KUKA KRL program: ab_st600_r1.src, ab_st600_r1.dat

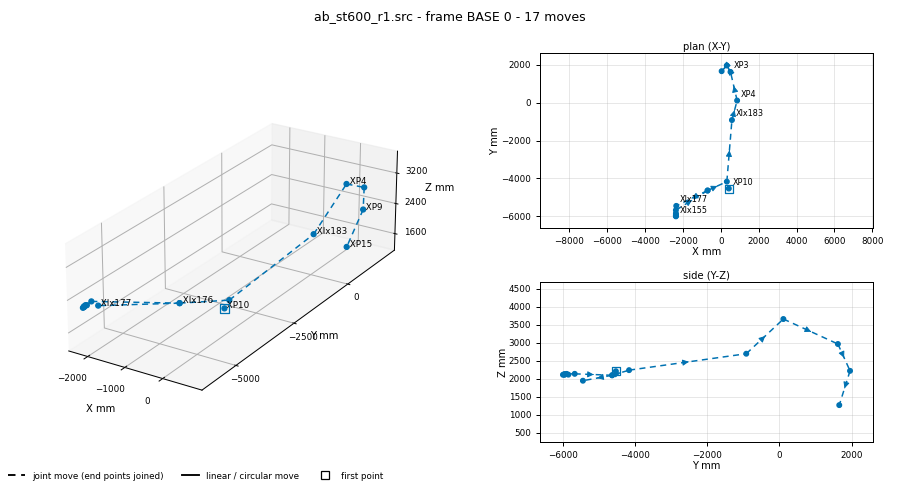
[picture p0: tool path of ab_st600_r1.src in frame BASE 0, 17 of 22 moves have a stored position in this frame; points joined in program order, loops and branches not executed]
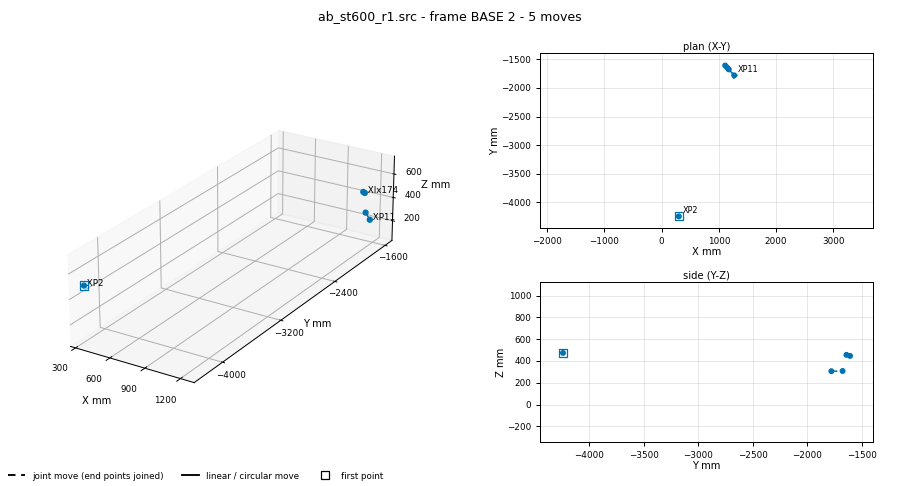
[picture p1: tool path of ab_st600_r1.src in frame BASE 2, 5 of 22 moves have a stored position in this frame; points joined in program order, loops and branches not executed]
--- ab_st600_r1.src ---
&ACCESS RVP1
&REL 63
&COMMENT Deposita traseira ACCELO
&PARAM DISKPATH = KRC:\R1\Program\MANIPULACAO LTC
&PARAM TEMPLATE = C:\KRC\Roboter\Template\vorgabe
&PARAM EDITMASK = *
DEF ab_st600_r1( )
;FOLD INI
  ;FOLD BASISTECH INI
    GLOBAL INTERRUPT DECL 3 WHEN $STOPMESS==TRUE DO IR_STOPM ( )
    INTERRUPT ON 3
    BAS (#INITMOV,0 )
  ;ENDFOLD (BASISTECH INI)
;FOLD GRIPPERTECH INI
USER_GRP(0,DUMMY,DUMMY,GDEFAULT)
;ENDFOLD (GRIPPERTECH INI)
  ;FOLD USER INI
    ;Make your modifications here

  ;ENDFOLD (USER INI)
;ENDFOLD (INI)

; Caracterização dos meios de produção:
; Versão Atual:
; 08/06/2013 12:00 Name: P13.050-R1 CHANGES: Deposita Traseira
; Accelo na Geobox

chk_w7_wechs_ok ( )              ; CHECK GRIPPER TRASEIRO


;FOLD PTP P10 Vel=100 % PDAT30 Tool[7]:Painel Traseiro Accelo Base[0];%{PE}%R 8.2.20,%MKUKATPBASIS,%CMOVE,%VPTP,%P 1:PTP, 2:P10, 3:, 5:100, 7:PDAT30
$BWDSTART=FALSE
PDAT_ACT=PPDAT30
FDAT_ACT=FP10
BAS(#PTP_PARAMS,100)
PTP XP10
;ENDFOLD

;FOLD PTP P2 Vel=100 % PDAT20 Tool[7]:Painel Traseiro Accelo Base[2]:Accelo;%{PE}%R 8.2.20,%MKUKATPBASIS,%CMOVE,%VPTP,%P 1:PTP, 2:P2, 3:, 5:100, 7:PDAT20
$BWDSTART=FALSE
PDAT_ACT=PPDAT20
FDAT_ACT=FP2
BAS(#PTP_PARAMS,100)
PTP XP2
;ENDFOLD

;FOLD OUT 3346 'Entrega peça Geo box' State=TRUE ;%{PE}%R 8.2.20,%MKUKATPBASIS,%COUT,%VOUTX,%P 2:3346, 3:Entrega peça Geo box, 5:TRUE, 6:
$OUT[3346]=TRUE
;ENDFOLD
;FOLD WAIT FOR ( IN 3346 'Aguarda lib. Entregar peça Geo box' );%{PE}%R 8.2.20,%MKUKATPBASIS,%CEXT_WAIT_FOR,%VEXT_WAIT_FOR,%P 2:, 4:, 5:$IN, 6:3346, 7:Aguarda lib. Entregar peça Geo box, 9:
WAIT FOR  ( $IN[3346] )
;ENDFOLD
;FOLD OUT 3346 'Entrega peça Geo box' State=FALSE ;%{PE}%R 8.2.20,%MKUKATPBASIS,%COUT,%VOUTX,%P 2:3346, 3:Entrega peça Geo box, 5:FALSE, 6:
$OUT[3346]=FALSE
;ENDFOLD
;FOLD OUT 3344 'R1 entregou peça geo box' State=FALSE ;%{PE}%R 8.2.20,%MKUKATPBASIS,%COUT,%VOUTX,%P 2:3344, 3:R1 entregou peça geo box, 5:FALSE, 6:
$OUT[3344]=FALSE
;ENDFOLD

;FOLD Collision.Monitoring_AREA_5_On ;%{PE}%MKUKATPUSER
COLLSTOP( 11, 1 ) ;not Interrupt-Controlled
;ENDFOLD
;FOLD Collision.Monitoring_AREA_6_On ;%{PE}%MKUKATPUSER
COLLSTOP( 12, 1 ) ;not Interrupt-Controlled
;ENDFOLD

;FOLD OUT 3340 'AREA_CLEAR_AGV' State=FALSE ;%{PE}%R 8.2.20,%MKUKATPBASIS,%COUT,%VOUTX,%P 2:3340, 3:AREA_CLEAR_AGV, 5:FALSE, 6:
$OUT[3340]=FALSE
;ENDFOLD
;FOLD OUT 3348 'Fora area GEOBOX' State=FALSE ;%{PE}%R 8.2.20,%MKUKATPBASIS,%COUT,%VOUTX,%P 2:3348, 3:Fora area GEOBOX, 5:FALSE, 6:
$OUT[3348]=FALSE
;ENDFOLD

;FOLD PTP lx176 CONT Vel=100 % PDAT8 Tool[7]:Painel Traseiro Accelo Base[0];%{PE}%R 8.2.20,%MKUKATPBASIS,%CMOVE,%VPTP,%P 1:PTP, 2:lx176, 3:C_DIS, 5:100, 7:PDAT8
$BWDSTART=FALSE
PDAT_ACT=PPDAT8
FDAT_ACT=Flx176
BAS(#PTP_PARAMS,100)
PTP Xlx176 C_DIS
;ENDFOLD
;FOLD PTP lx177 CONT Vel=100 % PDAT9 Tool[7]:Painel Traseiro Accelo Base[0];%{PE}%R 8.2.20,%MKUKATPBASIS,%CMOVE,%VPTP,%P 1:PTP, 2:lx177, 3:C_DIS, 5:100, 7:PDAT9
$BWDSTART=FALSE
PDAT_ACT=PPDAT9
FDAT_ACT=Flx177
BAS(#PTP_PARAMS,100)
PTP Xlx177 C_DIS
;ENDFOLD

;FOLD PTP P11 Vel=100 % PDAT31 Tool[7]:Painel Traseiro Accelo Base[2]:Accelo;%{PE}%R 8.2.20,%MKUKATPBASIS,%CMOVE,%VPTP,%P 1:PTP, 2:P11, 3:, 5:100, 7:PDAT31
$BWDSTART=FALSE
PDAT_ACT=PPDAT31
FDAT_ACT=FP11
BAS(#PTP_PARAMS,100)
PTP XP11
;ENDFOLD




;FOLD PTP lx178 Vel=100 % PDAT10 Tool[7]:Painel Traseiro Accelo Base[2]:Accelo;%{PE}%R 8.2.20,%MKUKATPBASIS,%CMOVE,%VPTP,%P 1:PTP, 2:lx178, 3:, 5:100, 7:PDAT10
$BWDSTART=FALSE
PDAT_ACT=PPDAT10
FDAT_ACT=Flx178
BAS(#PTP_PARAMS,100)
PTP Xlx178
;ENDFOLD


;FOLD PTP lx179 CONT Vel=70 % PDAT11 Tool[7]:Painel Traseiro Accelo Base[0];%{PE}%R 8.2.20,%MKUKATPBASIS,%CMOVE,%VPTP,%P 1:PTP, 2:lx179, 3:C_DIS, 5:70, 7:PDAT11
$BWDSTART=FALSE
PDAT_ACT=PPDAT11
FDAT_ACT=Flx179
BAS(#PTP_PARAMS,70)
PTP Xlx179 C_DIS
;ENDFOLD

IF (NOT(GHOST())) THEN

;FOLD ; bloqueado na Folder;%{PE}%R 8.2.20,%MKUKATPBASIS,%CCOMMENT,%VNORMAL,%P 2:bloqueado  na  Folder
;ENDFOLD

ENDIF

;FOLD LIN lx174 CONT Vel=0.25 m/s CPDAT0 Tool[7]:Painel Traseiro Accelo Base[0];%{PE}%R 8.2.20,%MKUKATPBASIS,%CMOVE,%VLIN,%P 1:LIN, 2:lx174, 3:C_DIS C_DIS, 5:0.25, 7:CPDAT0
$BWDSTART=FALSE
LDAT_ACT=LCPDAT0
FDAT_ACT=Flx174
BAS(#CP_PARAMS,0.25)
LIN Xlx174 C_DIS C_DIS
;ENDFOLD
;FOLD LIN lx173 CONT Vel=0.25 m/s CPDAT1 Tool[7]:Painel Traseiro Accelo Base[0];%{PE}%R 8.2.20,%MKUKATPBASIS,%CMOVE,%VLIN,%P 1:LIN, 2:lx173, 3:C_DIS C_DIS, 5:0.25, 7:CPDAT1
$BWDSTART=FALSE
LDAT_ACT=LCPDAT1
FDAT_ACT=Flx173
BAS(#CP_PARAMS,0.25)
LIN Xlx173 C_DIS C_DIS
;ENDFOLD
;FOLD LIN P12 Vel=0.25 m/s CPDAT2 Tool[7]:Painel Traseiro Accelo Base[0];%{PE}%R 8.2.20,%MKUKATPBASIS,%CMOVE,%VLIN,%P 1:LIN, 2:P12, 3:, 5:0.25, 7:CPDAT2
$BWDSTART=FALSE
LDAT_ACT=LCPDAT2
FDAT_ACT=FP12
BAS(#CP_PARAMS,0.25)
LIN XP12
;ENDFOLD

;FOLD ; POSICAO DE DEPOSITO DA PECA NA GEOBOX;%{PE}%R 8.2.20,%MKUKATPBASIS,%CCOMMENT,%VNORMAL,%P 2:POSICAO  DE  DEPOSITO  DA  PECA  NA  GEOBOX
;ENDFOLD
;FOLD LIN lx155 Vel=0.25 m/s L_OLP3 Tool[7]:Painel Traseiro Accelo Base[0];%{PE}%R 8.2.20,%MKUKATPBASIS,%CMOVE,%VLIN,%P 1:LIN, 2:lx155, 3:, 5:0.25, 7:L_OLP3
$BWDSTART=FALSE
LDAT_ACT=LL_OLP3
FDAT_ACT=Flx155
BAS(#CP_PARAMS,0.25)
LIN Xlx155
;ENDFOLD

;FOLD OUT 249 'Y1VR_FECHA_Accelo' State=FALSE ;%{PE}%R 8.2.20,%MKUKATPBASIS,%COUT,%VOUTX,%P 2:249, 3:Y1VR_FECHA_Accelo, 5:FALSE, 6:
$OUT[249]=FALSE
;ENDFOLD
;FOLD OUT 250 'YIVR_ABRE_Accelo' State=TRUE ;%{PE}%R 8.2.20,%MKUKATPBASIS,%COUT,%VOUTX,%P 2:250, 3:YIVR_ABRE_Accelo, 5:TRUE, 6:
$OUT[250]=TRUE
;ENDFOLD
;FOLD WAIT FOR ( IN 245 'Z1.2 - Grampo Recuado - Accelo - Traseiro' ) AND ( IN 247 'Z1.1 - Grampo Recuado - Accelo - Traseiro' );%{PE}%R 8.2.20,%MKUKATPBASIS,%CEXT_WAIT_FOR,%VEXT_WAIT_FOR,%P 2:, 4:, 5:$IN, 6:245, 7:Z1.2 - Grampo Recuado - Accelo - Traseiro, 9:AND, 10:, 12:, 13:$IN, 14:247, 15:Z1.1 - Grampo Recuado - Accelo - Traseiro, 17:
WAIT FOR  ( $IN[245] ) AND ( $IN[247] )
;ENDFOLD
;FOLD Collision.Monitoring_3_Off . ;%{PE}%MKUKATPUSER
COLLSTOP( 3, 2+0 )
;ENDFOLD

;FOLD OUT 3349 'R1 pegou peça' State=FALSE ;%{PE}%R 8.2.20,%MKUKATPBASIS,%COUT,%VOUTX,%P 2:3349, 3:R1 pegou peça, 5:FALSE, 6:
$OUT[3349]=FALSE
;ENDFOLD
;FOLD OUT 3345 'Solicita lib sair da geo box' State=TRUE ;%{PE}%R 8.2.20,%MKUKATPBASIS,%COUT,%VOUTX,%P 2:3345, 3:Solicita lib sair da geo box, 5:TRUE, 6:
$OUT[3345]=TRUE
;ENDFOLD
;FOLD WAIT FOR ( IN 3344 'Aguarda lib sair geo box' );%{PE}%R 8.2.20,%MKUKATPBASIS,%CEXT_WAIT_FOR,%VEXT_WAIT_FOR,%P 2:, 4:, 5:$IN, 6:3344, 7:Aguarda lib sair geo box, 9:
WAIT FOR  ( $IN[3344] )
;ENDFOLD
;FOLD OUT 3345 'Solicita lib sair da geo box' State=FALSE ;%{PE}%R 8.2.20,%MKUKATPBASIS,%COUT,%VOUTX,%P 2:3345, 3:Solicita lib sair da geo box, 5:FALSE, 6:
$OUT[3345]=FALSE
;ENDFOLD


;FOLD OUT 255 'Liga_Magnetico_Accelo' State=FALSE ;%{PE}%R 8.2.20,%MKUKATPBASIS,%COUT,%VOUTX,%P 2:255, 3:Liga_Magnetico_Accelo, 5:FALSE, 6:
$OUT[255]=FALSE
;ENDFOLD
;FOLD WAIT Time=0.5 sec;%{PE}%R 8.2.20,%MKUKATPBASIS,%CWAIT,%VWAIT,%P 3:0.5
WAIT SEC 0.5
;ENDFOLD
;FOLD OUT 256 'Desliga_Magnetico_Accelo' State=TRUE ;%{PE}%R 8.2.20,%MKUKATPBASIS,%COUT,%VOUTX,%P 2:256, 3:Desliga_Magnetico_Accelo, 5:TRUE, 6:
$OUT[256]=TRUE
;ENDFOLD


;FOLD OUT 244 'Liga_Sugador_Accelo' State=FALSE ;%{PE}%R 8.2.20,%MKUKATPBASIS,%COUT,%VOUTX,%P 2:244, 3:Liga_Sugador_Accelo, 5:FALSE, 6:
$OUT[244]=FALSE
;ENDFOLD
;FOLD WAIT Time=0.5 sec;%{PE}%R 8.2.20,%MKUKATPBASIS,%CWAIT,%VWAIT,%P 3:0.5
WAIT SEC 0.5
;ENDFOLD
;FOLD PULSE 243 'Liga_Soprador_Accelo' State=TRUE Time=1 sec;%{PE}%R 8.2.20,%MKUKATPBASIS,%COUT,%VPULSE,%P 2:243, 3:Liga_Soprador_Accelo, 5:TRUE, 6:, 8:1
PULSE($OUT[243], TRUE,1)
;ENDFOLD





;FOLD LIN lx159 Vel=0.25 m/s L_OLP4 Tool[7]:Painel Traseiro Accelo Base[0];%{PE}%R 8.2.20,%MKUKATPBASIS,%CMOVE,%VLIN,%P 1:LIN, 2:lx159, 3:, 5:0.25, 7:L_OLP4
$BWDSTART=FALSE
LDAT_ACT=LL_OLP4
FDAT_ACT=Flx159
BAS(#CP_PARAMS,0.25)
LIN Xlx159
;ENDFOLD
;FOLD PTP P1 CONT Vel=70 % PDAT1 Tool[7]:Painel Traseiro Accelo Base[0];%{PE}%R 8.2.20,%MKUKATPBASIS,%CMOVE,%VPTP,%P 1:PTP, 2:P1, 3:C_DIS, 5:70, 7:PDAT1
$BWDSTART=FALSE
PDAT_ACT=PPDAT1
FDAT_ACT=FP1
BAS(#PTP_PARAMS,70)
PTP XP1 C_DIS
;ENDFOLD
;FOLD PTP lx180 CONT Vel=100 % PDAT12 Tool[7]:Painel Traseiro Accelo Base[0];%{PE}%R 8.2.20,%MKUKATPBASIS,%CMOVE,%VPTP,%P 1:PTP, 2:lx180, 3:C_DIS, 5:100, 7:PDAT12
$BWDSTART=FALSE
PDAT_ACT=PPDAT12
FDAT_ACT=Flx180
BAS(#PTP_PARAMS,100)
PTP Xlx180 C_DIS
;ENDFOLD
;FOLD PTP lx181 CONT Vel=100 % PDAT13 Tool[7]:Painel Traseiro Accelo Base[0];%{PE}%R 8.2.20,%MKUKATPBASIS,%CMOVE,%VPTP,%P 1:PTP, 2:lx181, 3:C_DIS, 5:100, 7:PDAT13
$BWDSTART=FALSE
PDAT_ACT=PPDAT13
FDAT_ACT=Flx181
BAS(#PTP_PARAMS,100)
PTP Xlx181 C_DIS
;ENDFOLD

;FOLD PTP P14 CONT Vel=100 % PDAT32 Tool[7]:Painel Traseiro Accelo Base[0];%{PE}%R 8.2.20,%MKUKATPBASIS,%CMOVE,%VPTP,%P 1:PTP, 2:P14, 3:C_DIS, 5:100, 7:PDAT32
$BWDSTART=FALSE
PDAT_ACT=PPDAT32
FDAT_ACT=FP14
BAS(#PTP_PARAMS,100)
PTP XP14 C_DIS
;ENDFOLD

;FOLD PTP lx184 Vel=100 % PDAT33 Tool[7]:Painel Traseiro Accelo Base[0];%{PE}%R 8.2.20,%MKUKATPBASIS,%CMOVE,%VPTP,%P 1:PTP, 2:lx184, 3:, 5:100, 7:PDAT33
$BWDSTART=FALSE
PDAT_ACT=PPDAT33
FDAT_ACT=Flx184
BAS(#PTP_PARAMS,100)
PTP Xlx184
;ENDFOLD

;FOLD OUT 3344 'R1 entregou peça geo box' State=TRUE ;%{PE}%R 8.2.20,%MKUKATPBASIS,%COUT,%VOUTX,%P 2:3344, 3:R1 entregou peça geo box, 5:TRUE, 6:
$OUT[3344]=TRUE
;ENDFOLD
;FOLD OUT 3348 'Fora area GEOBOX' State=TRUE ;%{PE}%R 8.2.20,%MKUKATPBASIS,%COUT,%VOUTX,%P 2:3348, 3:Fora area GEOBOX, 5:TRUE, 6:
$OUT[3348]=TRUE
;ENDFOLD

;FOLD Collision.Monitoring_AREA_6_Off . ;%{PE}%MKUKATPUSER
COLLSTOP( 12, 2+0 )
;ENDFOLD

;FOLD PTP lx183 CONT Vel=100 % PDAT15 Tool[7]:Painel Traseiro Accelo Base[0];%{PE}%R 8.2.20,%MKUKATPBASIS,%CMOVE,%VPTP,%P 1:PTP, 2:lx183, 3:C_DIS, 5:100, 7:PDAT15
$BWDSTART=FALSE
PDAT_ACT=PPDAT15
FDAT_ACT=Flx183
BAS(#PTP_PARAMS,100)
PTP Xlx183 C_DIS
;ENDFOLD
;FOLD PTP P4 CONT Vel=100 % PDAT22 Tool[7]:Painel Traseiro Accelo Base[0];%{PE}%R 8.2.20,%MKUKATPBASIS,%CMOVE,%VPTP,%P 1:PTP, 2:P4, 3:C_DIS, 5:100, 7:PDAT22
$BWDSTART=FALSE
PDAT_ACT=PPDAT22
FDAT_ACT=FP4
BAS(#PTP_PARAMS,100)
PTP XP4 C_DIS
;ENDFOLD
;FOLD PTP P3 CONT Vel=100 % PDAT21 Tool[7]:Painel Traseiro Accelo Base[0];%{PE}%R 8.2.20,%MKUKATPBASIS,%CMOVE,%VPTP,%P 1:PTP, 2:P3, 3:C_DIS, 5:100, 7:PDAT21
$BWDSTART=FALSE
PDAT_ACT=PPDAT21
FDAT_ACT=FP3
BAS(#PTP_PARAMS,100)
PTP XP3 C_DIS
;ENDFOLD

;FOLD PTP P9 CONT Vel=100 % PDAT29 Tool[7]:Painel Traseiro Accelo Base[0];%{PE}%R 8.2.20,%MKUKATPBASIS,%CMOVE,%VPTP,%P 1:PTP, 2:P9, 3:C_DIS, 5:100, 7:PDAT29
$BWDSTART=FALSE
PDAT_ACT=PPDAT29
FDAT_ACT=FP9
BAS(#PTP_PARAMS,100)
PTP XP9 C_DIS
;ENDFOLD


;FOLD OUT 250 'YIVR_ABRE_Accelo' State=FALSE ;%{PE}%R 8.2.20,%MKUKATPBASIS,%COUT,%VOUTX,%P 2:250, 3:YIVR_ABRE_Accelo, 5:FALSE, 6:
$OUT[250]=FALSE
;ENDFOLD
;FOLD OUT 251 'Y2VR_FECHA_Accelo_Bolha' State=FALSE ;%{PE}%R 8.2.20,%MKUKATPBASIS,%COUT,%VOUTX,%P 2:251, 3:Y2VR_FECHA_Accelo_Bolha, 5:FALSE, 6:
$OUT[251]=FALSE
;ENDFOLD
;FOLD OUT 253 'Y3VR_AVANCA_CILINDRO_Accelo/Bolha' State=FALSE ;%{PE}%R 8.2.20,%MKUKATPBASIS,%COUT,%VOUTX,%P 2:253, 3:Y3VR_AVANCA_CILINDRO_Accelo/Bolha, 5:FALSE, 6:
$OUT[253]=FALSE
;ENDFOLD
;FOLD OUT 256 'Desliga_Magnetico_Accelo' State=FALSE ;%{PE}%R 8.2.20,%MKUKATPBASIS,%COUT,%VOUTX,%P 2:256, 3:Desliga_Magnetico_Accelo, 5:FALSE, 6:
$OUT[256]=FALSE
;ENDFOLD



;FOLD PTP P15 CONT Vel=100 % PDAT34 Tool[7]:Painel Traseiro Accelo Base[0];%{PE}%R 8.2.20,%MKUKATPBASIS,%CMOVE,%VPTP,%P 1:PTP, 2:P15, 3:C_DIS, 5:100, 7:PDAT34
$BWDSTART=FALSE
PDAT_ACT=PPDAT34
FDAT_ACT=FP15
BAS(#PTP_PARAMS,100)
PTP XP15 C_DIS
;ENDFOLD
;FOLD OUT 3344 'R1 entregou peça geo box' State=FALSE ;%{PE}%R 8.2.20,%MKUKATPBASIS,%COUT,%VOUTX,%P 2:3344, 3:R1 entregou peça geo box, 5:FALSE, 6:
$OUT[3344]=FALSE
;ENDFOLD

END

--- ab_st600_r1.dat ---
&ACCESS RVP1
&REL 63
&COMMENT Deposita traseira ACCELO
&PARAM DISKPATH = KRC:\R1\Program\MANIPULACAO LTC
&PARAM TEMPLATE = C:\KRC\Roboter\Template\vorgabe
&PARAM EDITMASK = *
DEFDAT  ab_st600_r1
;FOLD EXTERNAL DECLARATIONS;%{PE}%MKUKATPBASIS,%CEXT,%VCOMMON,%P
;FOLD GRIPPERTECH EXT
EXT  H50 (INT  :IN,INT  :IN,INT  :IN,GRP_TYP  :IN )
;ENDFOLD (GRIPPERTECH EXT)
;FOLD SPOTTECH EXT

;ENDFOLD (SPOTTECH EXT)
;FOLD BASISTECH EXT;%{PE}%MKUKATPBASIS,%CEXT,%VEXT,%P
EXT  BAS (BAS_COMMAND  :IN,REAL  :IN )
DECL INT SUCCESS
;ENDFOLD (BASISTECH EXT)
;FOLD USER EXT;%{E}%MKUKATPUSER,%CEXT,%VEXT,%P
;Make your modifications here

;ENDFOLD (USER EXT)
;ENDFOLD (EXTERNAL DECLARATIONS)
DECL BASIS_SUGG_T LAST_BASIS={POINT1[] "P0                      ",POINT2[] "P0                      ",CP_PARAMS[] "CPDAT0                  ",PTP_PARAMS[] "PDAT0                   ",CONT[] "                        ",CP_VEL[] "2.0                     ",PTP_VEL[] " 100                    ",SYNC_PARAMS[] "SYNCDAT                 ",SPL_NAME[] "S0                      "}
DECL LDAT LL_OLP3={VEL 0.25,ACC 100.0,APO_DIST 0.0,APO_FAC 0.0}
DECL E6POS Xlx155={X -2364.39893,Y -6000.32617,Z 2111.17212,A -177.279205,B -89.6416931,C -92.2932205,S 6,T 18,E1 -4969.44922,E2 0.0,E3 0.0,E4 0.0,E5 0.0,E6 0.0}
DECL FDAT Flx155={TOOL_NO 7,BASE_NO 0,IPO_FRAME #BASE,POINT2[] " ",TQ_STATE FALSE}
DECL LDAT LL_OLP4={VEL 0.25,ACC 100.0,APO_DIST 0.0,APO_FAC 0.0}
DECL E6POS Xlx159={X -2364.63696,Y -5957.36816,Z 2113.78589,A -159.226501,B -89.5623779,C -110.410797,S 6,T 18,E1 -4969.44385,E2 0.0,E3 0.0,E4 0.0,E5 0.0,E6 0.0}
DECL FDAT Flx159={TOOL_NO 7,BASE_NO 0,IPO_FRAME #BASE,POINT2[] " ",TQ_STATE FALSE}
DECL GRP_SUGG_T LAST_GRP={NUMBER[] "5                       ",STATE[] "3                       ",PARAMS[] "GDAT3                   "}
DECL GRP_TYP GGDAT1={G_APO #NO,GRP_TIME 0.200000003,CTRL #OFF,DLY 0,DST 1}
DECL E6POS XLX173={X 1111.56006,Y -1608.89197,Z 446.615112,A 47.66679,B -89.6412201,C -92.2391663,S 6,T 18,E1 -4969.44922,E2 0.0,E3 0.0,E4 0.0,E5 0.0,E6 0.0}
DECL FDAT Flx173={TOOL_NO 7,BASE_NO 2,IPO_FRAME #BASE,POINT2[] " ",TQ_STATE FALSE}
DECL LDAT LCPDAT1={VEL 2.0,ACC 100.0,APO_DIST 100.0,APO_FAC 50.0,AXIS_VEL 100.0,AXIS_ACC 100.0,ORI_TYP #VAR,CIRC_TYP #BASE,JERK_FAC 50.0,GEAR_JERK 50.0,EXAX_IGN 0}
DECL GRP_TYP GGDAT2={G_APO #NO,GRP_TIME 0.200000003,CTRL #OFF,DLY 0,DST 1}
DECL GRP_TYP GGDAT3={G_APO #NO,GRP_TIME 0.200000003,CTRL #OFF,DLY 0,DST 1}
DECL E6POS XLX176={X -692.677124,Y -4637.4751,Z 2096.96191,A -65.6902466,B -76.7407532,C 173.750504,S 6,T 18,E1 -3804.729,E2 0.0,E3 0.0,E4 0.0,E5 0.0,E6 0.0}
DECL FDAT Flx176={TOOL_NO 7,BASE_NO 0,IPO_FRAME #BASE,POINT2[] " ",TQ_STATE FALSE}
DECL PDAT PPDAT8={VEL 100.0,ACC 100.0,APO_DIST 100.0,APO_MODE #CDIS}
DECL E6POS XLX177={X -2346.24512,Y -5447.48877,Z 1945.67297,A 0.0,B -89.9999771,C 89.999733,S 6,T 18,E1 -4543.29883,E2 0.0,E3 0.0,E4 0.0,E5 0.0,E6 0.0}
DECL FDAT Flx177={TOOL_NO 7,BASE_NO 0,IPO_FRAME #BASE,POINT2[] " ",TQ_STATE FALSE}
DECL PDAT PPDAT9={VEL 100.0,ACC 100.0,APO_DIST 100.0,APO_MODE #CDIS}
DECL E6POS XLX178={X 1174.302,Y -1677.17395,Z 308.082001,A 113.473099,B -89.691658,C -158.477707,S 6,T 18,E1 -4969.43408,E2 0.0,E3 0.0,E4 0.0,E5 0.0,E6 0.0}
DECL FDAT Flx178={TOOL_NO 7,BASE_NO 2,IPO_FRAME #BASE,POINT2[] " ",TQ_STATE FALSE}
DECL PDAT PPDAT10={VEL 100.0,ACC 100.0,APO_DIST 0.0,APO_MODE #CDIS}
DECL E6POS XLX179={X -2365.16699,Y -5850.93311,Z 2114.04199,A -144.472198,B -89.4127502,C -125.252502,S 6,T 18,E1 -4969.43701,E2 0.0,E3 0.0,E4 0.0,E5 0.0,E6 0.0}
DECL FDAT Flx179={TOOL_NO 7,BASE_NO 0,IPO_FRAME #BASE,POINT2[] " ",TQ_STATE FALSE}
DECL PDAT PPDAT11={VEL 100.0,ACC 100.0,APO_DIST 0.0,APO_MODE #CDIS}
DECL E6POS XLX180={X -2365.10791,Y -5899.65723,Z 2135.40503,A -144.427795,B -89.4126816,C -125.296501,S 6,T 18,E1 -4969.43799,E2 0.0,E3 0.0,E4 0.0,E5 0.0,E6 0.0}
DECL FDAT Flx180={TOOL_NO 7,BASE_NO 0,IPO_FRAME #BASE,POINT2[] " ",TQ_STATE FALSE}
DECL PDAT PPDAT12={VEL 100.0,ACC 100.0,APO_DIST 100.0,APO_MODE #CDIS}
DECL E6POS XLX181={X -2366.20093,Y -5674.63281,Z 2136.73901,A -144.430405,B -89.4129715,C -125.294296,S 6,T 18,E1 -4969.43896,E2 0.0,E3 0.0,E4 0.0,E5 0.0,E6 0.0}
DECL FDAT Flx181={TOOL_NO 7,BASE_NO 0,IPO_FRAME #BASE,POINT2[] " ",TQ_STATE FALSE}
DECL PDAT PPDAT13={VEL 100.0,ACC 100.0,APO_DIST 100.0,APO_MODE #CDIS}
DECL E6POS XLX182={X 323.305206,Y -4167.68213,Z 2238.50903,A 8.81354809,B -76.7102737,C 135.989594,S 6,T 18,E1 -3134.729,E2 0.0,E3 0.0,E4 0.0,E5 0.0,E6 0.0}
DECL FDAT Flx182={TOOL_NO 7,BASE_NO 0,IPO_FRAME #BASE,POINT2[] " ",TQ_STATE FALSE}
DECL PDAT PPDAT14={VEL 100.0,ACC 100.0,APO_DIST 100.0,APO_MODE #CDIS}
DECL E6POS XLX183={X 591.650391,Y -918.8573,Z 2694.11011,A 114.587196,B -75.356163,C -26.1469097,S 2,T 2,E1 424.345612,E2 0.0,E3 0.0,E4 0.0,E5 0.0,E6 0.0}
DECL FDAT Flx183={TOOL_NO 7,BASE_NO 0,IPO_FRAME #BASE,POINT2[] " ",TQ_STATE FALSE}
DECL PDAT PPDAT15={VEL 100.0,ACC 100.0,APO_DIST 100.0,APO_MODE #CDIS}
DECL E6POS XP2={X 301.369202,Y -4243.51904,Z 473.870514,A -56.4879189,B -77.8458862,C 48.6962509,S 6,T 18,E1 -2796.73096,E2 0.0,E3 0.0,E4 0.0,E5 0.0,E6 0.0}
DECL FDAT FP2={TOOL_NO 7,BASE_NO 2,IPO_FRAME #BASE,POINT2[] " ",TQ_STATE FALSE}
DECL PDAT PPDAT20={VEL 100.0,ACC 100.0,APO_DIST 100.0,APO_MODE #CDIS}
DECL E6POS XP3={X 516.011902,Y 1621.49805,Z 2963.49805,A -103.589996,B -63.0337791,C -33.4023399,S 2,T 3,E1 424.345398,E2 0.0,E3 0.0,E4 0.0,E5 0.0,E6 0.0}
DECL FDAT FP3={TOOL_NO 7,BASE_NO 0,IPO_FRAME #BASE,POINT2[] " ",TQ_STATE FALSE}
DECL PDAT PPDAT21={VEL 100.0,ACC 100.0,APO_DIST 100.0,APO_MODE #CDIS}
DECL E6POS XP4={X 865.822388,Y 109.914597,Z 3656.11792,A -178.399597,B -34.341259,C -38.3228111,S 2,T 3,E1 424.345398,E2 0.0,E3 0.0,E4 0.0,E5 0.0,E6 0.0}
DECL FDAT FP4={TOOL_NO 7,BASE_NO 0,IPO_FRAME #BASE,POINT2[] " ",TQ_STATE FALSE}
DECL PDAT PPDAT22={VEL 100.0,ACC 100.0,APO_DIST 100.0,APO_MODE #CDIS}
DECL PDAT PPDAT29={VEL 100.0,ACC 100.0,APO_DIST 100.0,APO_MODE #CDIS}
DECL E6POS XP9={X 320.157104,Y 1957.98499,Z 2219.09204,A 78.0421066,B -89.2650528,C 159.536407,S 2,T 3,E1 47.2499619,E2 0.0,E3 0.0,E4 0.0,E5 0.0,E6 0.0}
DECL FDAT FP9={TOOL_NO 7,BASE_NO 0,IPO_FRAME #BASE,POINT2[] " ",TQ_STATE FALSE}
DECL E6POS XP10={X 427.052094,Y -4533.16895,Z 2209.23096,A -73.5140305,B -78.8540268,C -161.541,S 6,T 18,E1 -2536.18311,E2 0.0,E3 0.0,E4 0.0,E5 0.0,E6 0.0}
DECL FDAT FP10={TOOL_NO 7,BASE_NO 0,IPO_FRAME #BASE,POINT2[] " ",TQ_STATE FALSE}
DECL PDAT PPDAT30={VEL 100.0,ACC 80.0,APO_DIST 100.0,APO_MODE #CDIS}
DECL E6POS XP11={X 1268.90002,Y -1780.18201,Z 306.232208,A 113.343002,B -89.7930298,C -158.341797,S 6,T 18,E1 -4829.35889,E2 0.0,E3 0.0,E4 0.0,E5 0.0,E6 0.0}
DECL FDAT FP11={TOOL_NO 7,BASE_NO 2,IPO_FRAME #BASE,POINT2[] " ",TQ_STATE FALSE}
DECL PDAT PPDAT31={VEL 100.0,ACC 100.0,APO_DIST 100.0,APO_MODE #CDIS}
DECL E6POS XP12={X -2364.20898,Y -5965.22119,Z 2114.70703,A -179.8405,B -89.5075912,C -89.8852997,S 6,T 18,E1 -4969.44922,E2 0.0,E3 0.0,E4 0.0,E5 0.0,E6 0.0}
DECL FDAT FP12={TOOL_NO 7,BASE_NO 0,IPO_FRAME #BASE,POINT2[] " ",TQ_STATE FALSE}
DECL LDAT LCPDAT2={VEL 2.0,ACC 100.0,APO_DIST 100.0,APO_FAC 50.0,AXIS_VEL 100.0,AXIS_ACC 100.0,ORI_TYP #VAR,CIRC_TYP #BASE,JERK_FAC 50.0,GEAR_JERK 50.0,EXAX_IGN 0}
DECL E6POS XP13={X -2366.91309,Y -5901.98193,Z 2118.14307,A -131.508698,B -89.5476379,C -137.690903,S 6,T 18,E1 -4969.43604,E2 0.0,E3 0.0,E4 0.0,E5 0.0,E6 0.0}
DECL FDAT FP13={TOOL_NO 7,BASE_NO 0,IPO_FRAME #BASE,POINT2[] " ",TQ_STATE FALSE}
DECL LDAT LCPDAT3={VEL 2.0,ACC 100.0,APO_DIST 100.0,APO_FAC 50.0,AXIS_VEL 100.0,AXIS_ACC 100.0,ORI_TYP #VAR,CIRC_TYP #BASE,JERK_FAC 50.0,GEAR_JERK 50.0,EXAX_IGN 0}
DECL E6POS XP14={X -692.677673,Y -4637.4751,Z 2096.95996,A -65.689537,B -76.740593,C 173.749802,S 6,T 18,E1 -3804.729,E2 0.0,E3 0.0,E4 0.0,E5 0.0,E6 0.0}
DECL FDAT FP14={TOOL_NO 7,BASE_NO 0,IPO_FRAME #BASE,POINT2[] " ",TQ_STATE FALSE}
DECL PDAT PPDAT32={VEL 100.0,ACC 100.0,APO_DIST 100.0,APO_MODE #CDIS}
DECL PDAT PPDAT33={VEL 100.0,ACC 100.0,APO_DIST 100.0,APO_MODE #CDIS}
DECL E6POS Xlx184={X 323.305206,Y -4167.68213,Z 2238.50903,A 8.81354809,B -76.7102737,C 135.989594,S 6,T 18,E1 -3134.729,E2 0.0,E3 0.0,E4 0.0,E5 0.0,E6 0.0}
DECL FDAT Flx184={TOOL_NO 7,BASE_NO 0,IPO_FRAME #BASE,POINT2[] " ",TQ_STATE FALSE}
DECL E6POS XP15={X 48.8478699,Y 1659.33105,Z 1269.35205,A 78.5208435,B -58.8224716,C 169.365601,S 2,T 3,E1 -326.278107,E2 0.0,E3 0.0,E4 0.0,E5 0.0,E6 0.0}
DECL FDAT FP15={TOOL_NO 7,BASE_NO 0,IPO_FRAME #BASE,POINT2[] " ",TQ_STATE FALSE}
DECL PDAT PPDAT34={VEL 100.0,ACC 100.0,APO_DIST 100.0,APO_MODE #CDIS}
DECL LDAT LCPDAT0={VEL 2.0,ACC 100.0,APO_DIST 100.0,APO_FAC 50.0,AXIS_VEL 100.0,AXIS_ACC 100.0,ORI_TYP #VAR,CIRC_TYP #BASE,JERK_FAC 50.0,GEAR_JERK 50.0,EXAX_IGN 0}
DECL E6POS Xlx174={X 1143.54797,Y -1641.83203,Z 456.325012,A 64.9152374,B -89.5681381,C -109.548698,S 6,T 18,E1 -4969.44189,E2 0.0,E3 0.0,E4 0.0,E5 0.0,E6 0.0}
DECL FDAT Flx174={TOOL_NO 7,BASE_NO 2,IPO_FRAME #BASE,POINT2[] " ",TQ_STATE FALSE}
DECL E6POS XP1={X -2364.63696,Y -5957.36816,Z 2129.70703,A -159.2341,B -89.5623016,C -110.403297,S 6,T 18,E1 -4969.44385,E2 0.0,E3 0.0,E4 0.0,E5 0.0,E6 0.0}
DECL FDAT FP1={TOOL_NO 7,BASE_NO 0,IPO_FRAME #BASE,POINT2[] " ",TQ_STATE FALSE}
DECL PDAT PPDAT1={VEL 100.0,ACC 100.0,APO_DIST 0.0,APO_MODE #CDIS}
ENDDAT
